Omron CX-Programmer project NuevoProyecto (CX-Programmer 9.61)

# PLC NuevoPLC1: CQM1 CPU41

## Program NuevoPrograma1 (no task)
Local symbols
KM1 100.00 BOOL  ; Contactor arranque directo
LA 100.02 BOOL
LF 100.01 BOOL
PM 0.00 BOOL  ; Pulsador de marcha
PP 0.01 BOOL  ; Pulsador de paro
RT 0.02 BOOL  ; Contacto Relé Térmico

### Section Sección1

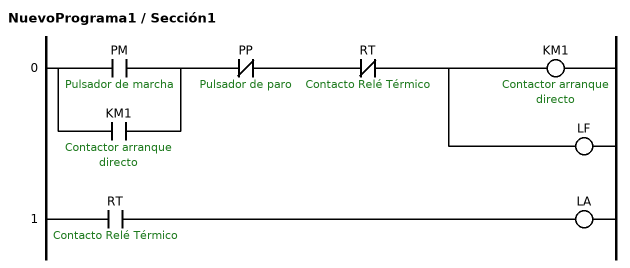
; rung 0
LD PM  ; Pulsador de marcha
OR KM1  ; Contactor arranque directo
ANDNOT PP  ; Pulsador de paro
ANDNOT RT  ; Contacto Relé Térmico
OUT KM1  ; Contactor arranque directo
OUT LF
; rung 1
LD RT  ; Contacto Relé Térmico
OUT LA

### Section END
; rung 0
END(01)